(*
Base interface for all FsControllerToolbox components.

Extends ``__SYSTEM.IQueryInterface`` to allow runtime type checking via
``__QUERYINTERFACE``.
*)
INTERFACE I_Component EXTENDS __SYSTEM.IQueryInterface

END_INTERFACE

(* stored: Version 1.1.0.1, ProductVersion 3.1.4024.15
   Itf I_Component: Id {2906025a-fa25-4a72-827e-2d345efa1901} *)
